// TIA Portal V21 export
// export: Created 2026-09-06T16:24:03.1416293Z, ExportSetting WithDefaults, DisplayName Totally Integrated Automation Portal, DisplayVersion V21 Hotfix 1, DisplayName STEP 7 Professional, DisplayVersion V21, DisplayName STEP 7 CFC, DisplayVersion V21, DisplayName STEP 7 Safety, DisplayVersion V21, DisplayName Tech WebApplication, DisplayVersion V21, DisplayName WinCC Basic/Comfort/Advanced, DisplayVersion V21, DisplayName SIMATIC Visualization Architect, DisplayVersion V21, DisplayName WinCC Unified, DisplayVersion V21, DisplayName SIMATIC Visualization Architect, DisplayVersion V21
DATA_BLOCK "DB_LinhaCompactador"   // DB1
VERSION : 0.1
// stored: AutoNumber true, DBAccessibleFromOPCUA true, InstanceOfName FB_LinhaCompactador, InstanceOfType FB
"FB_LinhaCompactador"
   // VAR
   //    T_Start_M6 { S7_SetPoint := 'True'} : TON_TIME;
   //    T_Start_M5 { S7_SetPoint := 'True'} : TON_TIME;
   //    T_Start_M34 { S7_SetPoint := 'True'} : TON_TIME;
   //    T_Stop_M12 { S7_SetPoint := 'True'} : TON_TIME;
   //    T_Stop_M34 { S7_SetPoint := 'True'} : TON_TIME;
   //    T_Stop_M5 { S7_SetPoint := 'True'} : TON_TIME;
   // END_VAR
BEGIN
END_DATA_BLOCK
